TYPE "TAx_DriveInterface"
VERSION : 0.1
// Block: TAx_DriveInterface
   STRUCT
      Infeed_ON : Bool;
      AccessPoint : HW_IO;
      AxisID : USInt;
      TokenChain : Int;
   END_STRUCT;

END_TYPE
